// TIA Portal V15.1 export
// export: Created 2024-06-21T08:41:02.0781303Z, ExportSetting WithDefaults, DisplayName Totally Integrated Automation Portal, DisplayVersion V15.1 Update 5, DisplayName TIA Portal Openness, DisplayVersion V15.1 Update 5, DisplayName SINAMICS Startdrive Advanced, DisplayVersion V15.1, DisplayName G130, G150, S120, S150, SINAMICS MV, S210, DisplayVersion V15.1, DisplayName G110M, G120, G120C, G120D, G120P, DisplayVersion V15.1, DisplayName STEP 7 Professional, DisplayVersion V15.1 Update 5, DisplayName STEP 7 Safety, DisplayVersion V15.1, DisplayName WinCC Professional, DisplayVersion V15.1 Update 5, DisplayName SIMATIC Visualization Architect, DisplayVersion V15.1
FUNCTION_BLOCK "LMovFnc3Pos2S"   // FB2192, FBD
TITLE = LMovFnc3Pos2S
{ S7_Optimized_Access := 'TRUE' }
VERSION : 0.1
// =============================================================================
// This module will be used for the steering of a three Position movement wit 2 speed
// It will get the commands from different Modes, evaluate the status of the 
// Interlock and give the command to the Actuator or direct to simple outputs.
// =============================================================================
// stored: AutoNumber false, IsIECCheckEnabled false, IsRetainMemResEnabled false, MemoryReserve 100, SetENOAutomatically False, UDAEnableTagReadback false
   VAR_INPUT
      I_Pos1 { ExternalAccessible := 'False'; ExternalVisible := 'False'; ExternalWritable := 'False'} : Bool;   // Position 1 Detection or Summary
      I_Pos2 { ExternalAccessible := 'False'; ExternalVisible := 'False'; ExternalWritable := 'False'} : Bool;   // Position 2 Detection or Summary
      I_Pos3 { ExternalAccessible := 'False'; ExternalVisible := 'False'; ExternalWritable := 'False'} : Bool;   // Position 3 Detection or Summary
      I_SlowPos1 { ExternalAccessible := 'False'; ExternalVisible := 'False'; ExternalWritable := 'False'} : Bool;   // Slow Position 1 Detection
      I_SlowPos2 { ExternalAccessible := 'False'; ExternalVisible := 'False'; ExternalWritable := 'False'} : Bool;   // Slow Position 2 Detection
      I_SlowPos3 { ExternalAccessible := 'False'; ExternalVisible := 'False'; ExternalWritable := 'False'} : Bool;   // Slow Position 3 Detection
      I_PBSet { ExternalAccessible := 'False'; ExternalVisible := 'False'; ExternalWritable := 'False'} : Bool;   // Push button for Set direction (used in manual with button OP panels )
      I_PBReset { ExternalAccessible := 'False'; ExternalVisible := 'False'; ExternalWritable := 'False'} : Bool;   // Push button for Reset direction (used in manual with Pushbutton OP panels)
      I_Pos1Begin { ExternalAccessible := 'False'; ExternalVisible := 'False'; ExternalWritable := 'False'} : Bool;   // Request Pos 1 Function Begin
      I_Pos2Begin { ExternalAccessible := 'False'; ExternalVisible := 'False'; ExternalWritable := 'False'} : Bool;   // Request Pos 2 Function Begin
      I_Pos3Begin { ExternalAccessible := 'False'; ExternalVisible := 'False'; ExternalWritable := 'False'} : Bool;   // Request Pos 3 Function Begin
      I_SetIntlkOK { ExternalAccessible := 'False'; ExternalVisible := 'False'; ExternalWritable := 'False'} : Bool;   // Interlock Set Ok
      I_ResIntlkOK { ExternalAccessible := 'False'; ExternalVisible := 'False'; ExternalWritable := 'False'} : Bool;   // Interlock Reset Ok
      I_SafetyOk { ExternalAccessible := 'False'; ExternalVisible := 'False'; ExternalWritable := 'False'} : Bool;   // Safety ok
      I_HardwareOk { ExternalAccessible := 'False'; ExternalVisible := 'False'; ExternalWritable := 'False'} : Bool;   // Safety Ok / Hardware Ok
   END_VAR
   VAR_OUTPUT
      O_CmdSetHighSpeed { ExternalAccessible := 'False'; ExternalVisible := 'False'; ExternalWritable := 'False'} : Bool;   // Command to Activate Set movement
      O_CmdResHighSpeed { ExternalAccessible := 'False'; ExternalVisible := 'False'; ExternalWritable := 'False'} : Bool;   // Command to Activate Reset movement
      O_CmdSetLowSpeed { ExternalAccessible := 'False'; ExternalVisible := 'False'; ExternalWritable := 'False'} : Bool;   // Command to Activate Slow Set movement
      O_CmdResLowSpeed { ExternalAccessible := 'False'; ExternalVisible := 'False'; ExternalWritable := 'False'} : Bool;   // Command to Activate Slow Reset movement
      O_CmdPos1 { ExternalAccessible := 'False'; ExternalVisible := 'False'; ExternalWritable := 'False'} : Bool;   // Command to activate Set movement / Command to Activate Pos1 movement
      O_CmdPos2 { ExternalAccessible := 'False'; ExternalVisible := 'False'; ExternalWritable := 'False'} : Bool;   // Command to activate Set movement / Command to Activate Pos2 movement
      O_CmdPos3 { ExternalAccessible := 'False'; ExternalVisible := 'False'; ExternalWritable := 'False'} : Bool;   // Command to activate Reset movement / Command to Activate Pos3 movement
      O_FuncRunning { ExternalAccessible := 'False'; ExternalVisible := 'False'; ExternalWritable := 'False'} : Bool;   // Signal that the function is running
      O_FuncBusyTM { ExternalAccessible := 'False'; ExternalVisible := 'False'; ExternalWritable := 'False'} : Bool;   // Memory Signal that the function is busy
      O_Pos1Finished { ExternalAccessible := 'False'; ExternalVisible := 'False'; ExternalWritable := 'False'} : Bool;   // Position1 Finished
      O_Pos2Finished { ExternalAccessible := 'False'; ExternalVisible := 'False'; ExternalWritable := 'False'} : Bool;   // Position2 Finished
      O_Pos3Finished { ExternalAccessible := 'False'; ExternalVisible := 'False'; ExternalWritable := 'False'} : Bool;   // Position3 Finished
      O_IntlkSetAlm { ExternalAccessible := 'False'; ExternalVisible := 'False'; ExternalWritable := 'False'} : Bool;   // Alarm Interlock Set
      O_IntlkResAlm { ExternalAccessible := 'False'; ExternalVisible := 'False'; ExternalWritable := 'False'} : Bool;   // Alarm Interlock Reset
      O_FuncIsSelInMan { ExternalAccessible := 'False'; ExternalVisible := 'False'; ExternalWritable := 'False'} : Bool;   // The function is Selected in manual Mode
      O_LED { ExternalAccessible := 'False'; ExternalVisible := 'False'; ExternalWritable := 'False'} : Bool;   // LED - Indication
      O_AlarmABCondition { ExternalAccessible := 'False'; ExternalVisible := 'False'; ExternalWritable := 'False'} : Bool;   // Alarms AB condition
   END_VAR
   VAR_IN_OUT
      IO_Modes : "Modes";   // Modes
      H_HMI : "H_HMI";   // Animation
      H_MovFnc3Pos2S : "H_MovFnc3Pos";   // Animation
      H_FncSelInHMI { ExternalAccessible := 'False'; ExternalVisible := 'False'; ExternalWritable := 'False'} : Bool;   // This function is Selected to run from HMI
      C_AlarmResetUsed { ExternalAccessible := 'False'; ExternalVisible := 'False'; ExternalWritable := 'False'} : Bool;   // If true, the alrms will be stored untill Reseted
      C_EnableMemBegin { ExternalAccessible := 'False'; ExternalVisible := 'False'; ExternalWritable := 'False'} : Bool;   // Enable memory Begin (Command request is memorised until pos reached)
      C_EnIntlkAlm { ExternalAccessible := 'False'; ExternalVisible := 'False'; ExternalWritable := 'False'} : Bool := TRUE;   // Enable Interlock Alarm
      C_ForceManual { ExternalAccessible := 'False'; ExternalVisible := 'False'; ExternalWritable := 'False'} : Bool := FALSE;   // Force Manual
   END_VAR
   VAR
      ResetAlarm { ExternalAccessible := 'False'; ExternalVisible := 'False'; ExternalWritable := 'False'} : Bool;   // Reset Alarm Memory
      BeginPos1Req { ExternalAccessible := 'False'; ExternalVisible := 'False'; ExternalWritable := 'False'} : Bool;   // Request Pos 1 Function Begin
      BeginPos2Req { ExternalAccessible := 'False'; ExternalVisible := 'False'; ExternalWritable := 'False'} : Bool;   // Request Pos 2 Function Begin
      BeginPos3Req { ExternalAccessible := 'False'; ExternalVisible := 'False'; ExternalWritable := 'False'} : Bool;   // Request Pos 3 Function Begin
      CmdSet { ExternalAccessible := 'False'; ExternalVisible := 'False'; ExternalWritable := 'False'} : Bool;   // Command set
      CmdSetSl { ExternalAccessible := 'False'; ExternalVisible := 'False'; ExternalWritable := 'False'} : Bool;   // Command to Activate Slow Set movement
      CmdSetRequest { ExternalAccessible := 'False'; ExternalVisible := 'False'; ExternalWritable := 'False'} : Bool;   // Set Command request to Activate the Interlock
      CmdRes { ExternalAccessible := 'False'; ExternalVisible := 'False'; ExternalWritable := 'False'} : Bool;   // Command Reset
      CmdResSl { ExternalAccessible := 'False'; ExternalVisible := 'False'; ExternalWritable := 'False'} : Bool;   // Command to Activate Slow Reset movement
      CmdResRequest { ExternalAccessible := 'False'; ExternalVisible := 'False'; ExternalWritable := 'False'} : Bool;   // Reset Command request to Activate the Interlock
   END_VAR
   VAR RETAIN
      BetweenPos1Pos2 { ExternalAccessible := 'False'; ExternalVisible := 'False'; ExternalWritable := 'False'} : Bool;   // Table Between Pos 1 And 2
      BetweenPos1Pos2Set { ExternalAccessible := 'False'; ExternalVisible := 'False'; ExternalWritable := 'False'} : Bool;   // Table Between Pos 1 And 2 Set
      BetweenPos1Pos2Res { ExternalAccessible := 'False'; ExternalVisible := 'False'; ExternalWritable := 'False'} : Bool;   // Table Between Pos 1 And 2 Reset
      BetweenPos2Pos3 { ExternalAccessible := 'False'; ExternalVisible := 'False'; ExternalWritable := 'False'} : Bool;   // Table Between Pos 2 And 3
      BetweenPos2Pos3Set { ExternalAccessible := 'False'; ExternalVisible := 'False'; ExternalWritable := 'False'} : Bool;   // Table Between Pos 2 And 3 Set
      BetweenPos2Pos3Res { ExternalAccessible := 'False'; ExternalVisible := 'False'; ExternalWritable := 'False'} : Bool;   // Table Between Pos 2 And 3 Reset
   END_VAR
   VAR
      Pos2SetReached { ExternalAccessible := 'False'; ExternalVisible := 'False'; ExternalWritable := 'False'} : Bool;   // Position 2 Set Reached
      P_CmdSetRequest { ExternalAccessible := 'False'; ExternalVisible := 'False'; ExternalWritable := 'False'} : Bool;   // Cmd Request Set Pos Trig
      Pos2ResReached { ExternalAccessible := 'False'; ExternalVisible := 'False'; ExternalWritable := 'False'} : Bool;   // Position 2 Reset Reached
      P_CmdResRequest { ExternalAccessible := 'False'; ExternalVisible := 'False'; ExternalWritable := 'False'} : Bool;   // Cmd Request Res Pos Trig
      CmdPos1 { ExternalAccessible := 'False'; ExternalVisible := 'False'; ExternalWritable := 'False'} : Bool;   // Command to activate Set movement / Command to Activate Pos1 movement
      CmdPos2 { ExternalAccessible := 'False'; ExternalVisible := 'False'; ExternalWritable := 'False'} : Bool;   // Command to activate Set movement / Command to Activate Pos2 movement
      CmdPos3 { ExternalAccessible := 'False'; ExternalVisible := 'False'; ExternalWritable := 'False'} : Bool;   // Command to activate Reset movement / Command to Activate Pos3 movement
      IntlkSetAlm { ExternalAccessible := 'False'; ExternalVisible := 'False'; ExternalWritable := 'False'} : Bool;   // Alarm Interlock Set
      IntlkResAlm { ExternalAccessible := 'False'; ExternalVisible := 'False'; ExternalWritable := 'False'} : Bool;   // Alarm Interlock Reset
      IntlkSetAlmCond { ExternalAccessible := 'False'; ExternalVisible := 'False'; ExternalWritable := 'False'} : Bool;   // Alarm Interlock Set condition
      IntlkResAlmCond { ExternalAccessible := 'False'; ExternalVisible := 'False'; ExternalWritable := 'False'} : Bool;   // Alarm Interlock Reset condition
      FuncRunning { ExternalAccessible := 'False'; ExternalVisible := 'False'; ExternalWritable := 'False'} : Bool;   // Function is running
      FuncBusyTM { ExternalAccessible := 'False'; ExternalVisible := 'False'; ExternalWritable := 'False'} : Bool;   // Memory Signal that the function is busy
      Edge { ExternalAccessible := 'False'; ExternalVisible := 'False'; ExternalWritable := 'False'} : Array[1..5] of Bool;   // Edge
      AlarmTimer { ExternalAccessible := 'False'; ExternalVisible := 'False'; ExternalWritable := 'False'} : "LTimer";
      AlmFilterResult { ExternalAccessible := 'False'; ExternalVisible := 'False'; ExternalWritable := 'False'} : Bool;
   END_VAR
   VAR_TEMP   // added for the SCL form of the ladder/FBD networks
      _w1 : Bool;
      _w2 : Bool;
      _w3 : Bool;
      _w4 : Bool;
   END_VAR
BEGIN

REGION Network 1: **** 2.2 - Alarms - Alarm Generation **** Alarm Filter
   // Alarm Filter
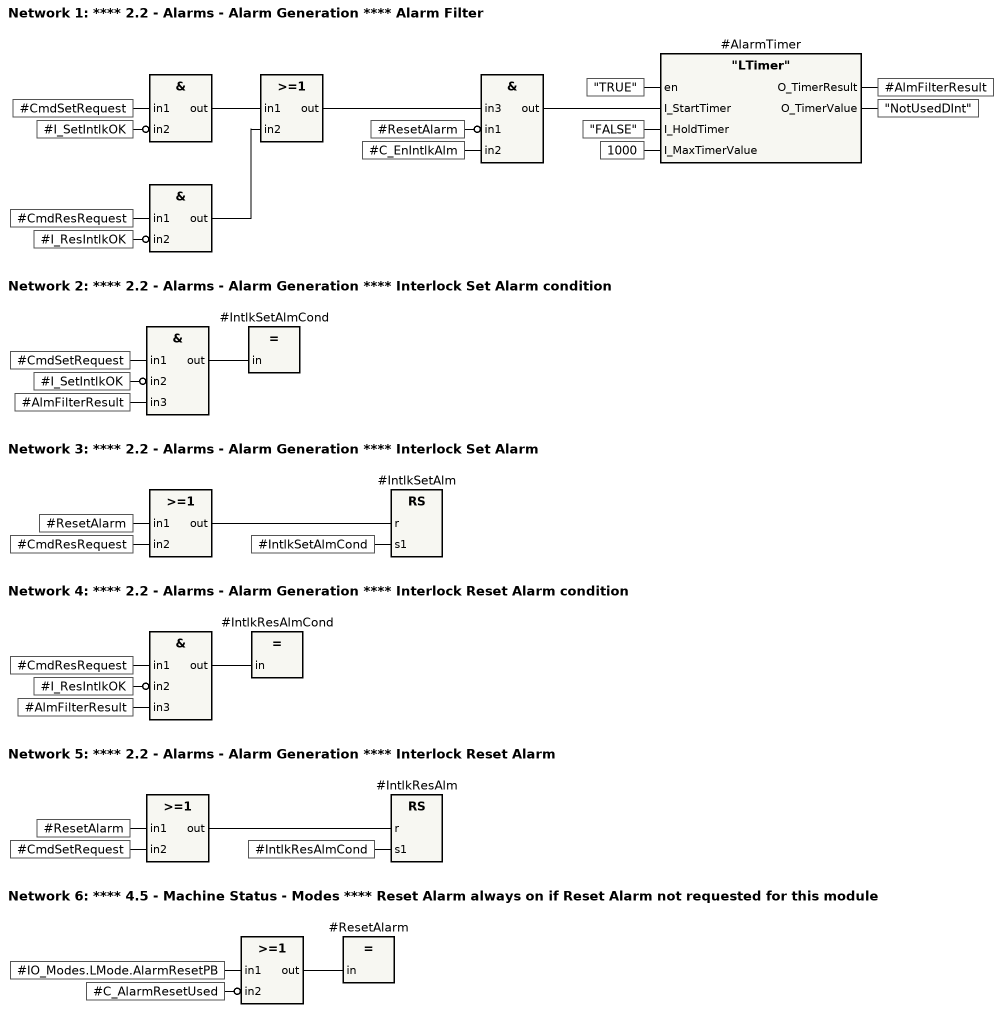
   IF "TRUE" THEN
       #AlarmTimer(I_StartTimer := ((#CmdSetRequest AND NOT #I_SetIntlkOK) OR (#CmdResRequest AND NOT #I_ResIntlkOK)) AND NOT #ResetAlarm AND #C_EnIntlkAlm,   // "LTimer"
                   I_HoldTimer := "FALSE",
                   I_MaxTimerValue := 1000,
                   O_TimerResult => #AlmFilterResult,
                   O_TimerValue => "NotUsedDInt");
   END_IF;
END_REGION

REGION Network 2: **** 2.2 - Alarms - Alarm Generation **** Interlock Set Alarm condition
   // Interlock Set Alarm condition
   #IntlkSetAlmCond := #CmdSetRequest AND NOT #I_SetIntlkOK AND #AlmFilterResult;
END_REGION

REGION Network 3: **** 2.2 - Alarms - Alarm Generation **** Interlock Set Alarm
   // Interlock Set Alarm
   IF #ResetAlarm OR #CmdResRequest THEN
       #IntlkSetAlm := FALSE;   // RS flip-flop
   END_IF;
   IF #IntlkSetAlmCond THEN #IntlkSetAlm := TRUE; END_IF;
END_REGION

REGION Network 4: **** 2.2 - Alarms - Alarm Generation **** Interlock Reset Alarm condition
   // Interlock Reset Alarm condition
   #IntlkResAlmCond := #CmdResRequest AND NOT #I_ResIntlkOK AND #AlmFilterResult;
END_REGION

REGION Network 5: **** 2.2 - Alarms - Alarm Generation **** Interlock Reset Alarm
   // Interlock Reset Alarm
   IF #ResetAlarm OR #CmdSetRequest THEN
       #IntlkResAlm := FALSE;   // RS flip-flop
   END_IF;
   IF #IntlkResAlmCond THEN #IntlkResAlm := TRUE; END_IF;
END_REGION

REGION Network 6: **** 4.5 - Machine Status - Modes **** Reset Alarm always on if Reset Alarm not requested for this module
   // Reset Alarm always on if Reset Alarm not requested for this module
   #ResetAlarm := #IO_Modes.LMode.AlarmResetPB OR NOT #C_AlarmResetUsed;
END_REGION

REGION Network 7: **** 4.6 - Machine Status - Indication **** Icon Animation
   // Icon Animation
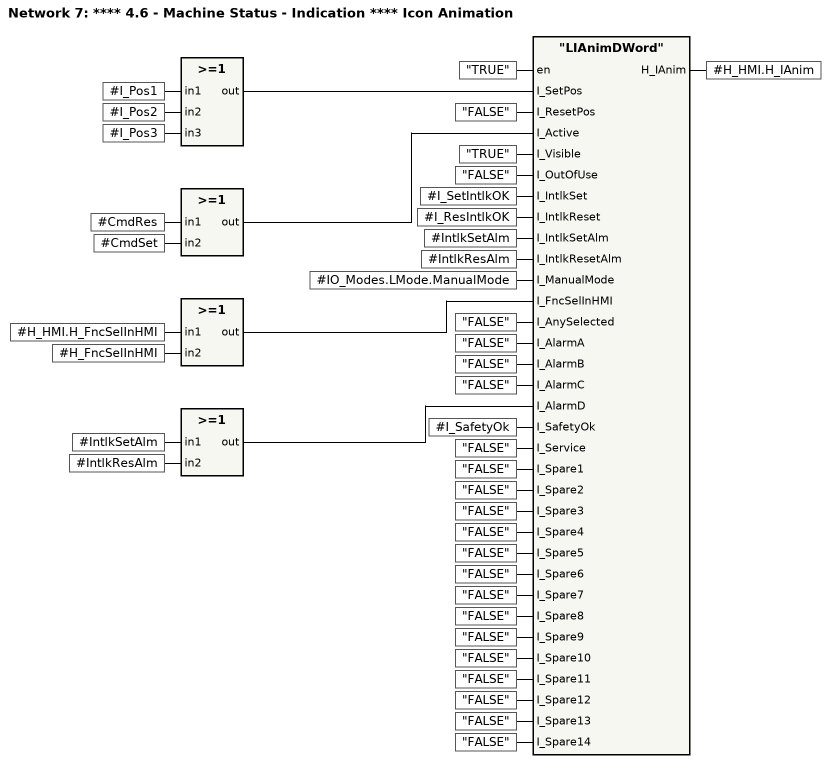
   IF "TRUE" THEN
       "LIAnimDWord"(I_SetPos := #I_Pos1 OR #I_Pos2 OR #I_Pos3,
                     I_ResetPos := "FALSE",
                     I_Active := #CmdRes OR #CmdSet,
                     I_Visible := "TRUE",
                     I_OutOfUse := "FALSE",
                     I_IntlkSet := #I_SetIntlkOK,
                     I_IntlkReset := #I_ResIntlkOK,
                     I_IntlkSetAlm := #IntlkSetAlm,
                     I_IntlkResetAlm := #IntlkResAlm,
                     I_ManualMode := #IO_Modes.LMode.ManualMode,
                     I_FncSelInHMI := #H_HMI.H_FncSelInHMI OR #H_FncSelInHMI,
                     I_AnySelected := "FALSE",
                     I_AlarmA := "FALSE",
                     I_AlarmB := "FALSE",
                     I_AlarmC := "FALSE",
                     I_AlarmD := #IntlkSetAlm OR #IntlkResAlm,
                     I_SafetyOk := #I_SafetyOk,
                     I_Service := "FALSE",
                     I_Spare1 := "FALSE",
                     I_Spare2 := "FALSE",
                     I_Spare3 := "FALSE",
                     I_Spare4 := "FALSE",
                     I_Spare5 := "FALSE",
                     I_Spare6 := "FALSE",
                     I_Spare7 := "FALSE",
                     I_Spare8 := "FALSE",
                     I_Spare9 := "FALSE",
                     I_Spare10 := "FALSE",
                     I_Spare11 := "FALSE",
                     I_Spare12 := "FALSE",
                     I_Spare13 := "FALSE",
                     I_Spare14 := "FALSE",
                     H_IAnim => #H_HMI.H_IAnim);
   END_IF;
END_REGION

REGION Network 8: **** 4.6 - Machine Status - Indication **** Animation
   // Animation
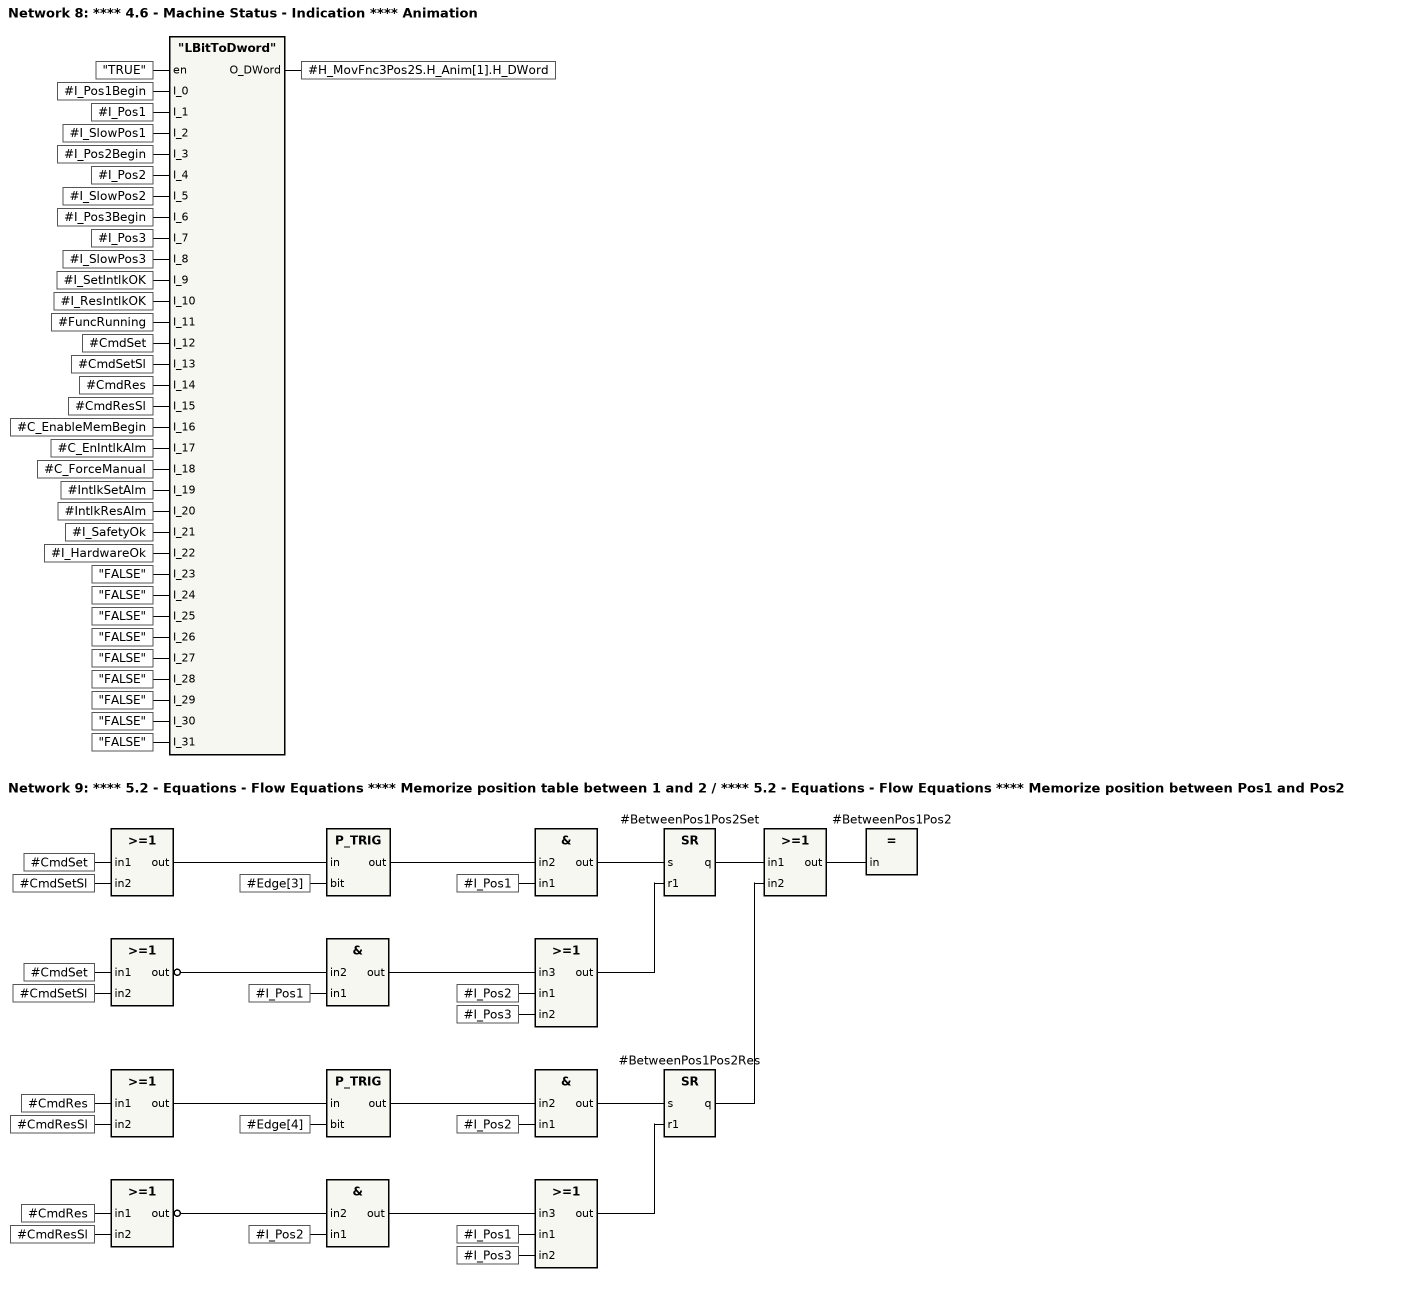
   IF "TRUE" THEN
       "LBitToDword"(I_0 := #I_Pos1Begin,
                     I_1 := #I_Pos1,
                     I_2 := #I_SlowPos1,
                     I_3 := #I_Pos2Begin,
                     I_4 := #I_Pos2,
                     I_5 := #I_SlowPos2,
                     I_6 := #I_Pos3Begin,
                     I_7 := #I_Pos3,
                     I_8 := #I_SlowPos3,
                     I_9 := #I_SetIntlkOK,
                     I_10 := #I_ResIntlkOK,
                     I_11 := #FuncRunning,
                     I_12 := #CmdSet,
                     I_13 := #CmdSetSl,
                     I_14 := #CmdRes,
                     I_15 := #CmdResSl,
                     I_16 := #C_EnableMemBegin,
                     I_17 := #C_EnIntlkAlm,
                     I_18 := #C_ForceManual,
                     I_19 := #IntlkSetAlm,
                     I_20 := #IntlkResAlm,
                     I_21 := #I_SafetyOk,
                     I_22 := #I_HardwareOk,
                     I_23 := "FALSE",
                     I_24 := "FALSE",
                     I_25 := "FALSE",
                     I_26 := "FALSE",
                     I_27 := "FALSE",
                     I_28 := "FALSE",
                     I_29 := "FALSE",
                     I_30 := "FALSE",
                     I_31 := "FALSE",
                     O_DWord => #H_MovFnc3Pos2S.H_Anim[1].H_DWord);
   END_IF;
END_REGION

REGION Network 9: **** 5.2 - Equations - Flow Equations **** Memorize position table between 1 and 2 / **** 5.2 - Equations - Flow Equations **** Memorize position between Pos1 and Pos2
   // Memorize Position table between 1 and 2
   #_w1 := #CmdSet OR #CmdSetSl;
   #_w2 := #_w1 AND NOT #Edge[3];   // rising edge
   #Edge[3] := #_w1;
   IF #_w2 AND #I_Pos1 THEN
       #BetweenPos1Pos2Set := TRUE;   // SR flip-flop
   END_IF;
   IF (NOT (#CmdSet OR #CmdSetSl) AND #I_Pos1) OR #I_Pos2 OR #I_Pos3 THEN
       #BetweenPos1Pos2Set := FALSE;
   END_IF;
   #_w3 := #CmdRes OR #CmdResSl;
   #_w4 := #_w3 AND NOT #Edge[4];   // rising edge
   #Edge[4] := #_w3;
   IF #_w4 AND #I_Pos2 THEN
       #BetweenPos1Pos2Res := TRUE;   // SR flip-flop
   END_IF;
   IF (NOT (#CmdRes OR #CmdResSl) AND #I_Pos2) OR #I_Pos1 OR #I_Pos3 THEN
       #BetweenPos1Pos2Res := FALSE;
   END_IF;
   #BetweenPos1Pos2 := #BetweenPos1Pos2Set OR #BetweenPos1Pos2Res;
END_REGION

REGION Network 10: **** 5.2 - Equations - Flow Equations **** Memorize position between 2 and 3 / **** 5.2 - Equations - Flow Equations **** Memorize position between Pos2 and Pos3
   // Memorize Position table  2 and 3
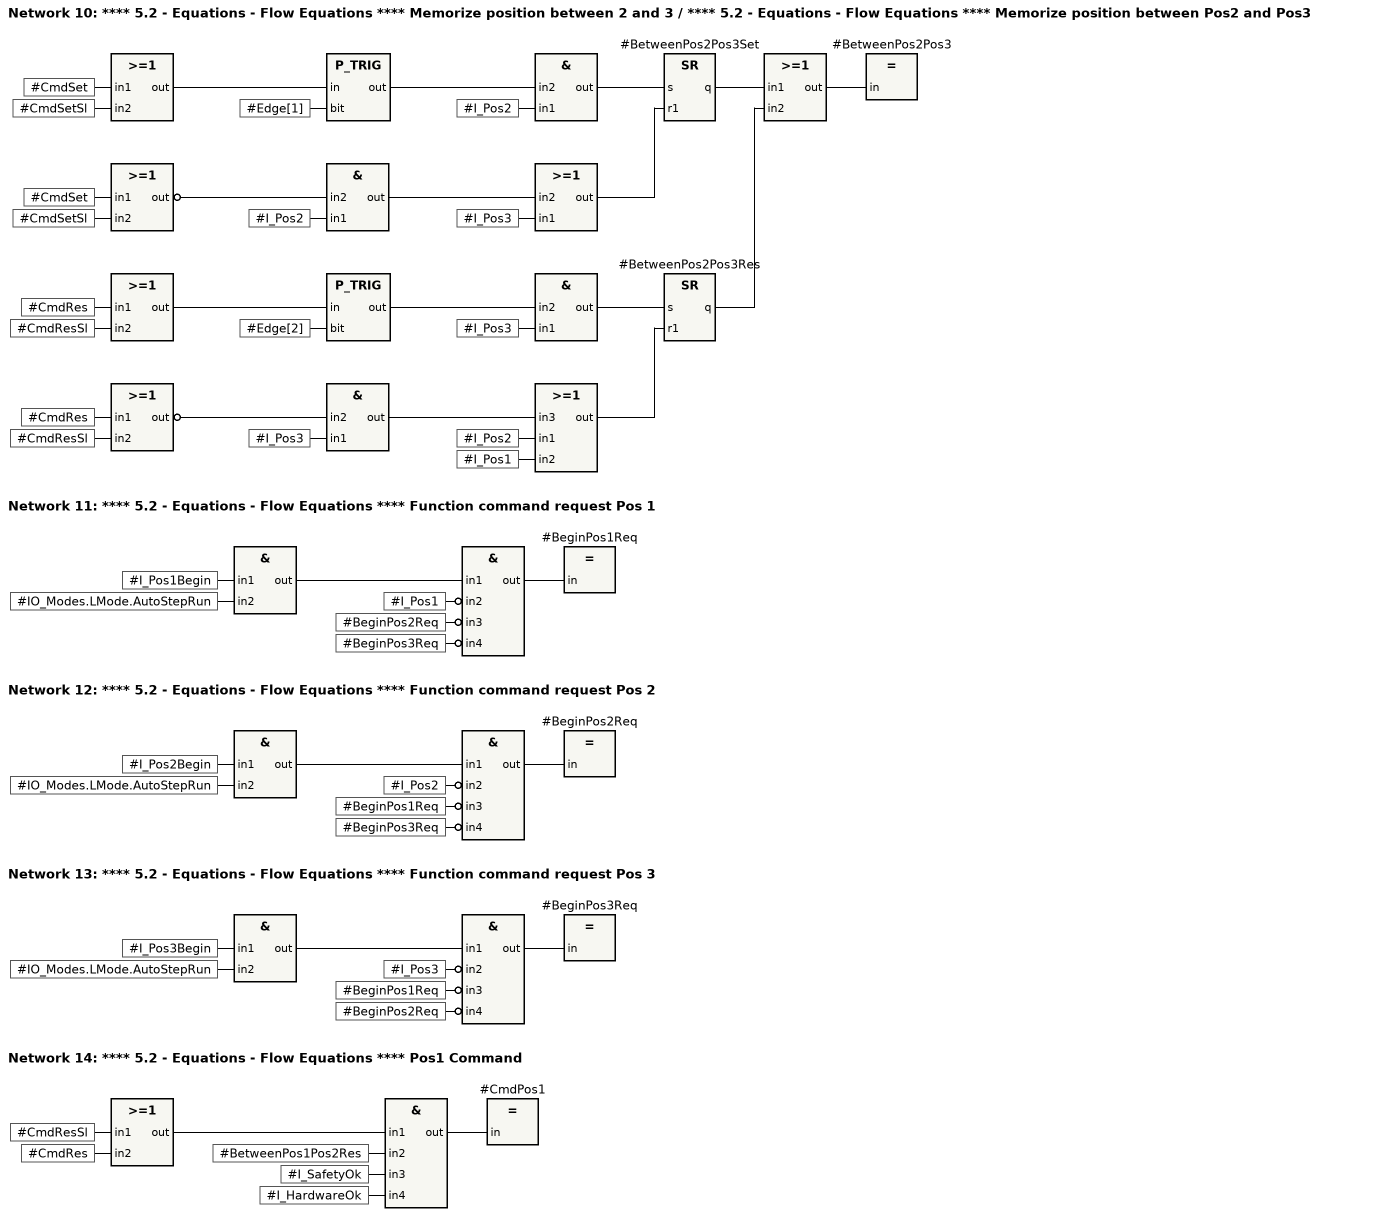
   #_w1 := #CmdSet OR #CmdSetSl;
   #_w2 := #_w1 AND NOT #Edge[1];   // rising edge
   #Edge[1] := #_w1;
   IF #_w2 AND #I_Pos2 THEN
       #BetweenPos2Pos3Set := TRUE;   // SR flip-flop
   END_IF;
   IF (NOT (#CmdSet OR #CmdSetSl) AND #I_Pos2) OR #I_Pos3 THEN #BetweenPos2Pos3Set := FALSE; END_IF;
   #_w3 := #CmdRes OR #CmdResSl;
   #_w4 := #_w3 AND NOT #Edge[2];   // rising edge
   #Edge[2] := #_w3;
   IF #_w4 AND #I_Pos3 THEN
       #BetweenPos2Pos3Res := TRUE;   // SR flip-flop
   END_IF;
   IF (NOT (#CmdRes OR #CmdResSl) AND #I_Pos3) OR #I_Pos2 OR #I_Pos1 THEN
       #BetweenPos2Pos3Res := FALSE;
   END_IF;
   #BetweenPos2Pos3 := #BetweenPos2Pos3Set OR #BetweenPos2Pos3Res;
END_REGION

REGION Network 11: **** 5.2 - Equations - Flow Equations **** Function command request Pos 1
   // Function command request Pos 1
   #BeginPos1Req := #I_Pos1Begin AND #IO_Modes.LMode.AutoStepRun AND NOT #I_Pos1 AND NOT #BeginPos2Req AND NOT #BeginPos3Req;
END_REGION

REGION Network 12: **** 5.2 - Equations - Flow Equations **** Function command request Pos 2
   // Function command request Pos 2
   #BeginPos2Req := #I_Pos2Begin AND #IO_Modes.LMode.AutoStepRun AND NOT #I_Pos2 AND NOT #BeginPos1Req AND NOT #BeginPos3Req;
END_REGION

REGION Network 13: **** 5.2 - Equations - Flow Equations **** Function command request Pos 3
   // Function command request Pos 3
   #BeginPos3Req := #I_Pos3Begin AND #IO_Modes.LMode.AutoStepRun AND NOT #I_Pos3 AND NOT #BeginPos1Req AND NOT #BeginPos2Req;
END_REGION

REGION Network 14: **** 5.2 - Equations - Flow Equations **** Pos1 Command
   // Pos1 Command
   #CmdPos1 := (#CmdResSl OR #CmdRes) AND #BetweenPos1Pos2Res AND #I_SafetyOk AND #I_HardwareOk;
END_REGION

REGION Network 15: **** 5.2 - Equations - Flow Equations **** Pos2 Command
   // Pos2 Command
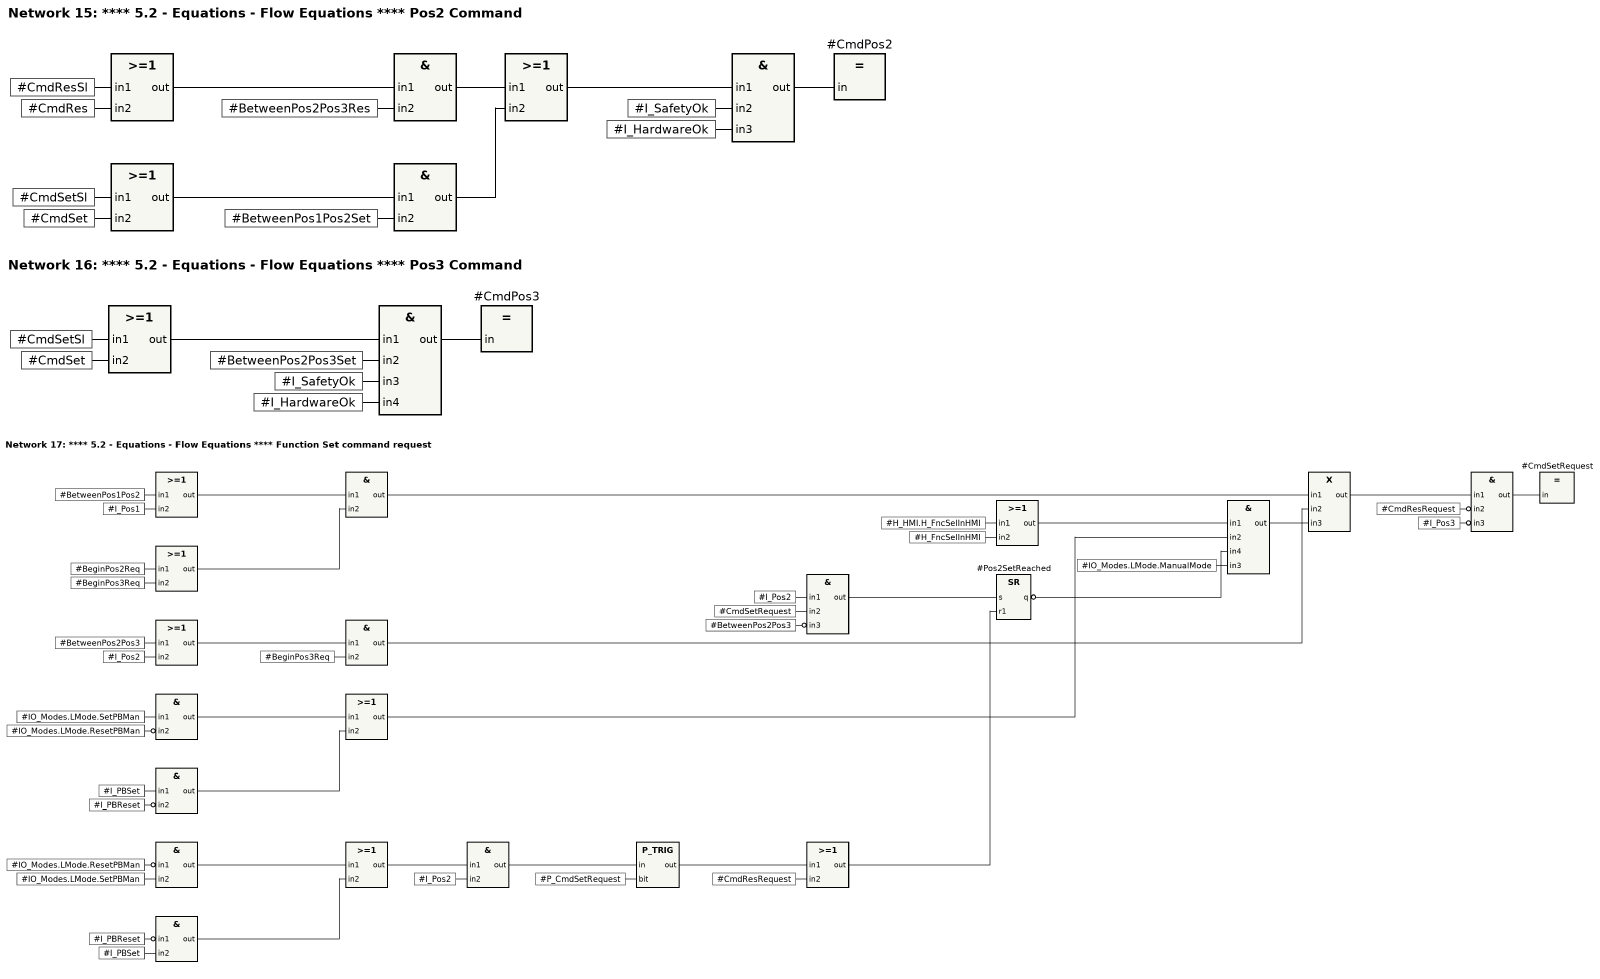
   #CmdPos2 := (((#CmdResSl OR #CmdRes) AND #BetweenPos2Pos3Res) OR ((#CmdSetSl OR #CmdSet) AND #BetweenPos1Pos2Set)) AND #I_SafetyOk AND #I_HardwareOk;
END_REGION

REGION Network 16: **** 5.2 - Equations - Flow Equations **** Pos3 Command
   // Pos3 Command
   #CmdPos3 := (#CmdSetSl OR #CmdSet) AND #BetweenPos2Pos3Set AND #I_SafetyOk AND #I_HardwareOk;
END_REGION

REGION Network 17: **** 5.2 - Equations - Flow Equations **** Function Set command request
   // Function Set command request
   #_w1 := ((NOT #IO_Modes.LMode.ResetPBMan AND #IO_Modes.LMode.SetPBMan) OR (NOT #I_PBReset AND #I_PBSet)) AND #I_Pos2;
   #_w2 := #_w1 AND NOT #P_CmdSetRequest;   // rising edge
   #P_CmdSetRequest := #_w1;
   IF #I_Pos2 AND #CmdSetRequest AND NOT #BetweenPos2Pos3 THEN
       #Pos2SetReached := TRUE;   // SR flip-flop
   END_IF;
   IF #_w2 OR #CmdResRequest THEN #Pos2SetReached := FALSE; END_IF;
   #CmdSetRequest := (((#BetweenPos1Pos2 OR #I_Pos1) AND (#BeginPos2Req OR #BeginPos3Req)) XOR ((#BetweenPos2Pos3 OR #I_Pos2) AND #BeginPos3Req) XOR ((#H_HMI.H_FncSelInHMI OR #H_FncSelInHMI) AND ((#IO_Modes.LMode.SetPBMan AND NOT #IO_Modes.LMode.ResetPBMan) OR (#I_PBSet AND NOT #I_PBReset)) AND NOT #Pos2SetReached AND #IO_Modes.LMode.ManualMode)) AND NOT #CmdResRequest AND NOT #I_Pos3;
END_REGION

REGION Network 18: **** 5.2 - Equations - Flow Equations **** Function Reset command request
   // Function Reset command request
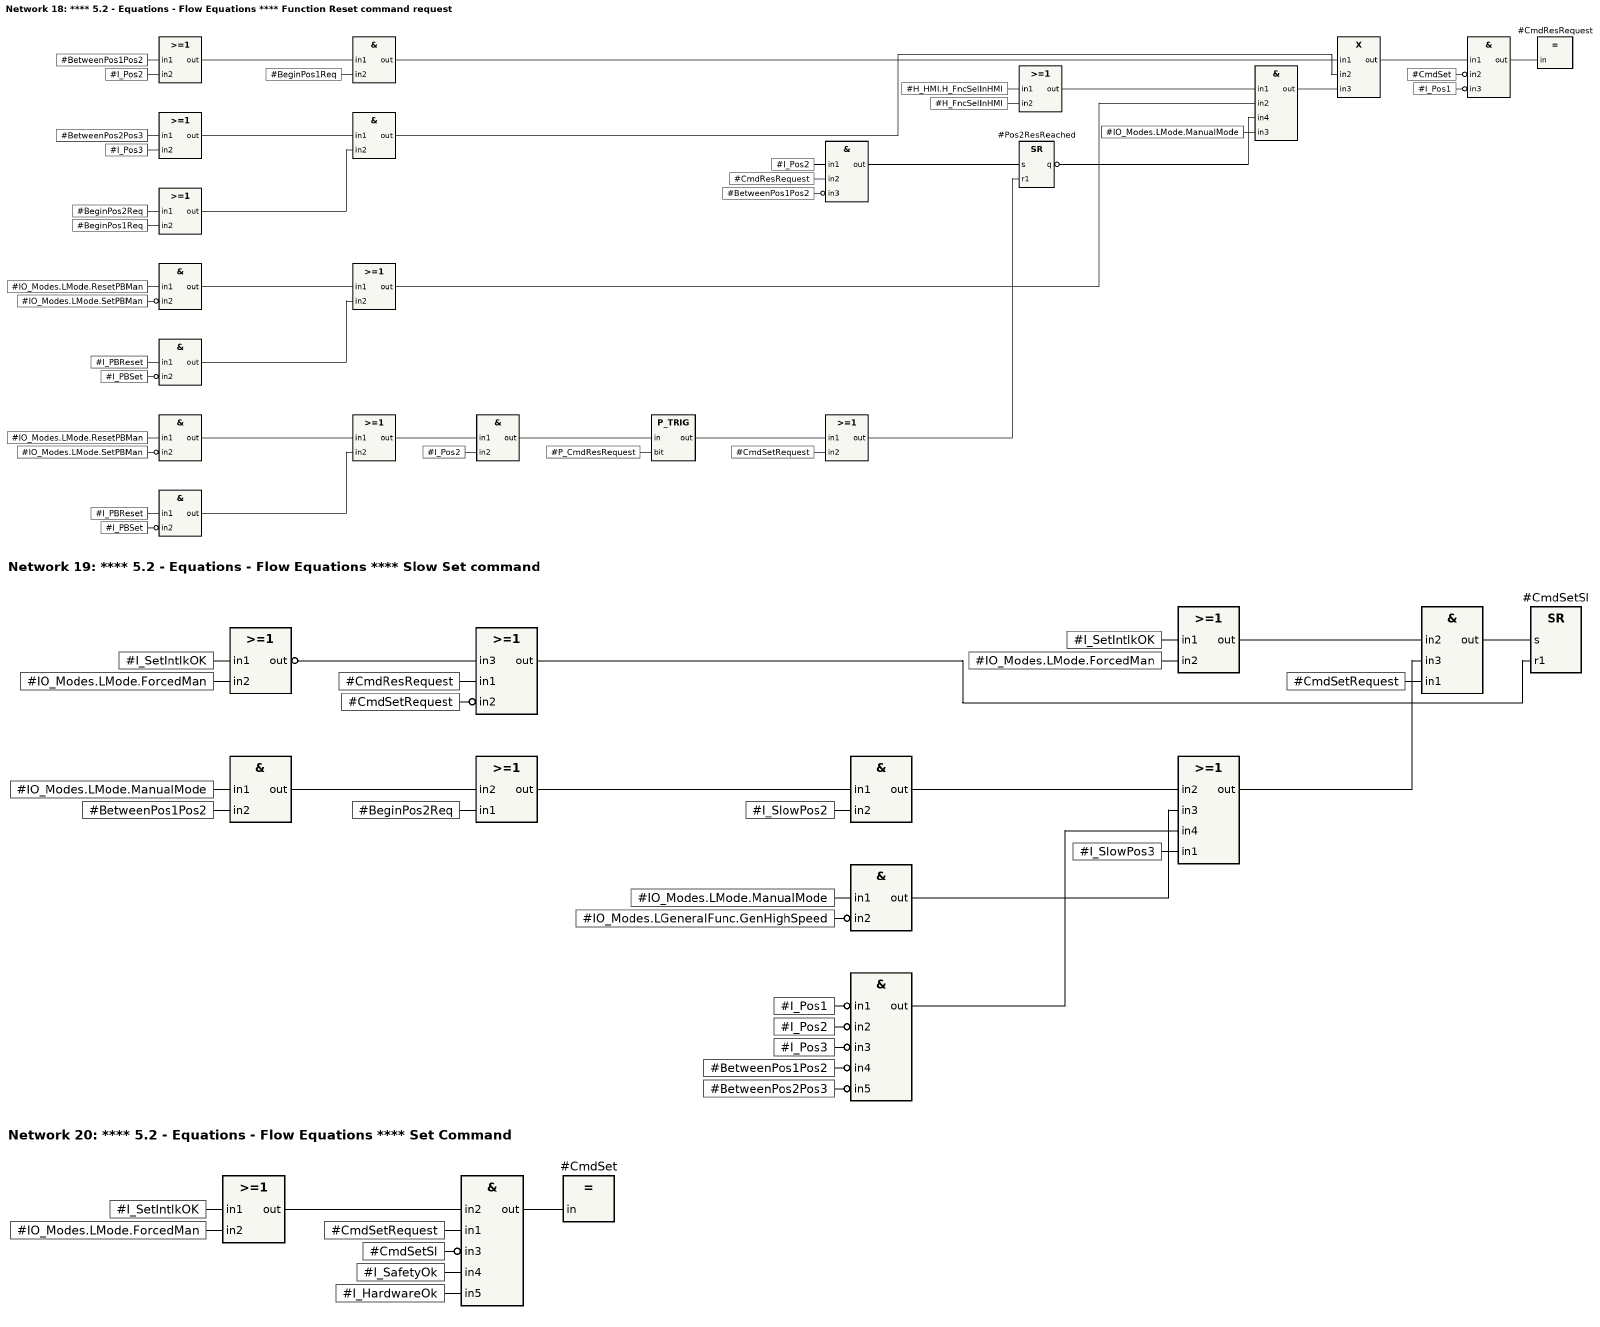
   #_w1 := ((#IO_Modes.LMode.ResetPBMan AND NOT #IO_Modes.LMode.SetPBMan) OR (#I_PBReset AND NOT #I_PBSet)) AND #I_Pos2;
   #_w2 := #_w1 AND NOT #P_CmdResRequest;   // rising edge
   #P_CmdResRequest := #_w1;
   IF #I_Pos2 AND #CmdResRequest AND NOT #BetweenPos1Pos2 THEN
       #Pos2ResReached := TRUE;   // SR flip-flop
   END_IF;
   IF #_w2 OR #CmdSetRequest THEN #Pos2ResReached := FALSE; END_IF;
   #CmdResRequest := (((#BetweenPos1Pos2 OR #I_Pos2) AND #BeginPos1Req) XOR ((#BetweenPos2Pos3 OR #I_Pos3) AND (#BeginPos2Req OR #BeginPos1Req)) XOR ((#H_HMI.H_FncSelInHMI OR #H_FncSelInHMI) AND ((#IO_Modes.LMode.ResetPBMan AND NOT #IO_Modes.LMode.SetPBMan) OR (#I_PBReset AND NOT #I_PBSet)) AND NOT #Pos2ResReached AND #IO_Modes.LMode.ManualMode)) AND NOT #CmdSet AND NOT #I_Pos1;
END_REGION

REGION Network 19: **** 5.2 - Equations - Flow Equations **** Slow Set command
   // Slow Set command
   IF (#I_SetIntlkOK OR #IO_Modes.LMode.ForcedMan) AND ((((#IO_Modes.LMode.ManualMode AND #BetweenPos1Pos2) OR #BeginPos2Req) AND #I_SlowPos2) OR (#IO_Modes.LMode.ManualMode AND NOT #IO_Modes.LGeneralFunc.GenHighSpeed) OR (NOT #I_Pos1 AND NOT #I_Pos2 AND NOT #I_Pos3 AND NOT #BetweenPos1Pos2 AND NOT #BetweenPos2Pos3) OR #I_SlowPos3) AND #CmdSetRequest THEN
       #CmdSetSl := TRUE;   // SR flip-flop
   END_IF;
   IF NOT (#I_SetIntlkOK OR #IO_Modes.LMode.ForcedMan) OR #CmdResRequest OR NOT #CmdSetRequest THEN
       #CmdSetSl := FALSE;
   END_IF;
END_REGION

REGION Network 20: **** 5.2 - Equations - Flow Equations **** Set Command
   // Set Command
   #CmdSet := (#I_SetIntlkOK OR #IO_Modes.LMode.ForcedMan) AND #CmdSetRequest AND NOT #CmdSetSl AND #I_SafetyOk AND #I_HardwareOk;
END_REGION

REGION Network 21: **** 5.2 - Equations - Flow Equations **** Slow Reset command
   // Slow Reset command
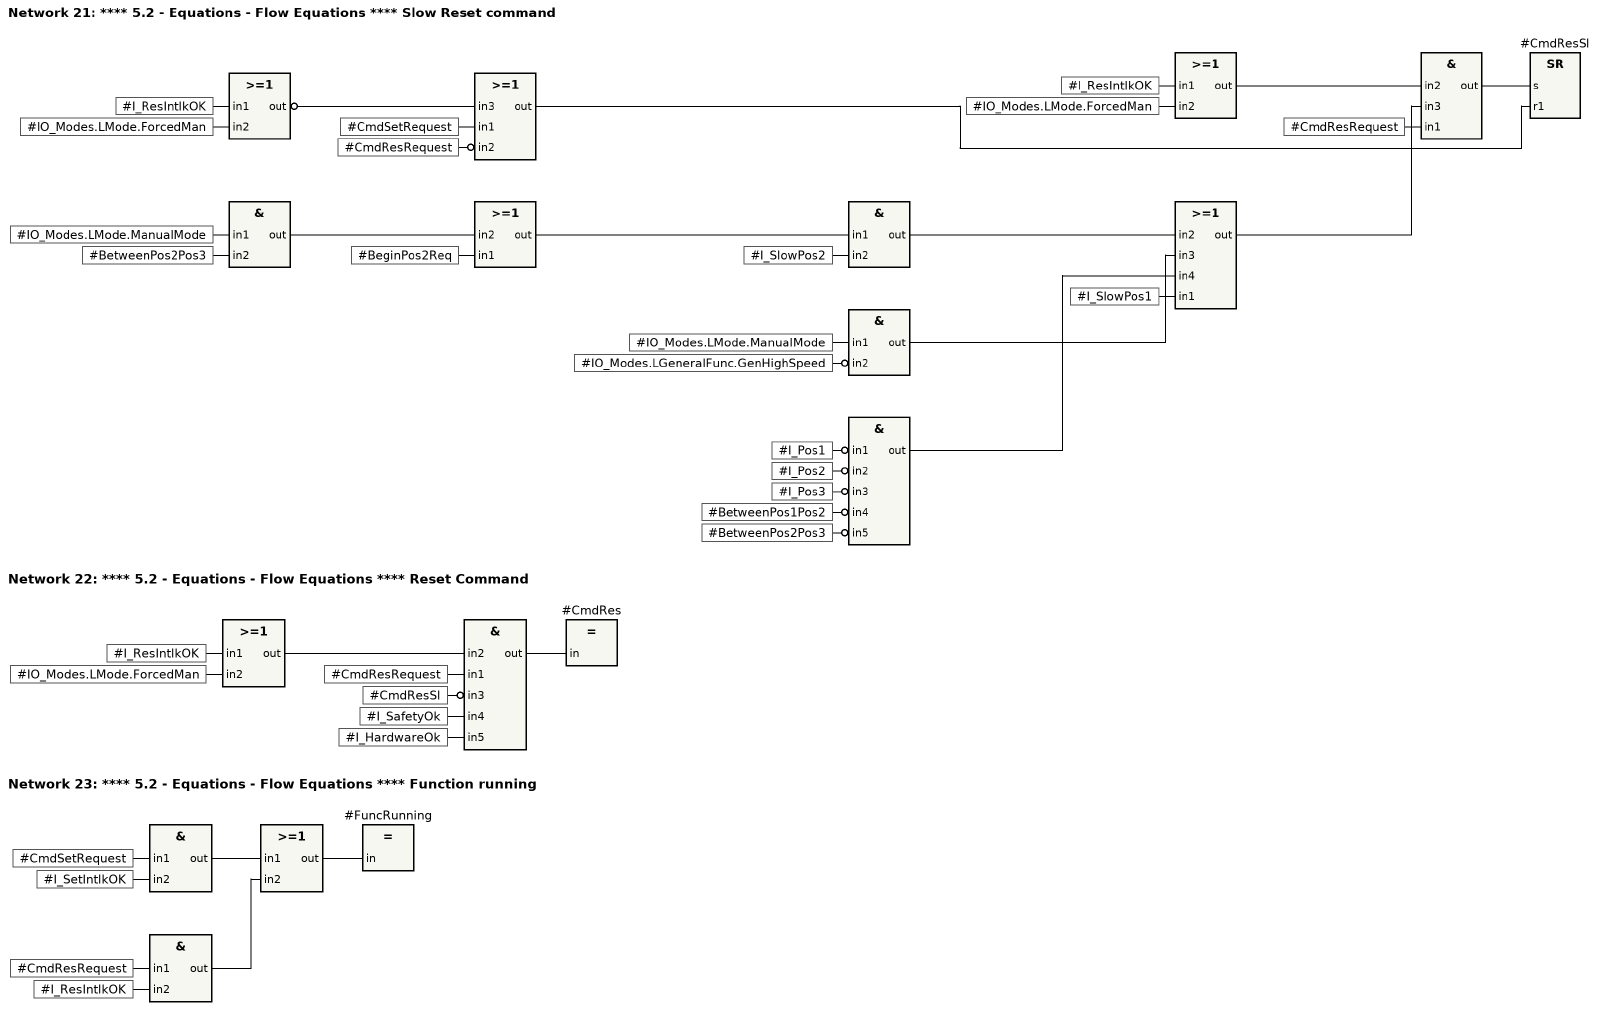
   IF (#I_ResIntlkOK OR #IO_Modes.LMode.ForcedMan) AND ((((#IO_Modes.LMode.ManualMode AND #BetweenPos2Pos3) OR #BeginPos2Req) AND #I_SlowPos2) OR (#IO_Modes.LMode.ManualMode AND NOT #IO_Modes.LGeneralFunc.GenHighSpeed) OR (NOT #I_Pos1 AND NOT #I_Pos2 AND NOT #I_Pos3 AND NOT #BetweenPos1Pos2 AND NOT #BetweenPos2Pos3) OR #I_SlowPos1) AND #CmdResRequest THEN
       #CmdResSl := TRUE;   // SR flip-flop
   END_IF;
   IF NOT (#I_ResIntlkOK OR #IO_Modes.LMode.ForcedMan) OR #CmdSetRequest OR NOT #CmdResRequest THEN
       #CmdResSl := FALSE;
   END_IF;
END_REGION

REGION Network 22: **** 5.2 - Equations - Flow Equations **** Reset Command
   // Reset Command
   #CmdRes := (#I_ResIntlkOK OR #IO_Modes.LMode.ForcedMan) AND #CmdResRequest AND NOT #CmdResSl AND #I_SafetyOk AND #I_HardwareOk;
END_REGION

REGION Network 23: **** 5.2 - Equations - Flow Equations **** Function running
   // Function running
   #FuncRunning := (#CmdSetRequest AND #I_SetIntlkOK) OR (#CmdResRequest AND #I_ResIntlkOK);
END_REGION

REGION Network 24: **** 5.2 - Equations - Flow Equations **** Set Function Running
   // Set Function Running
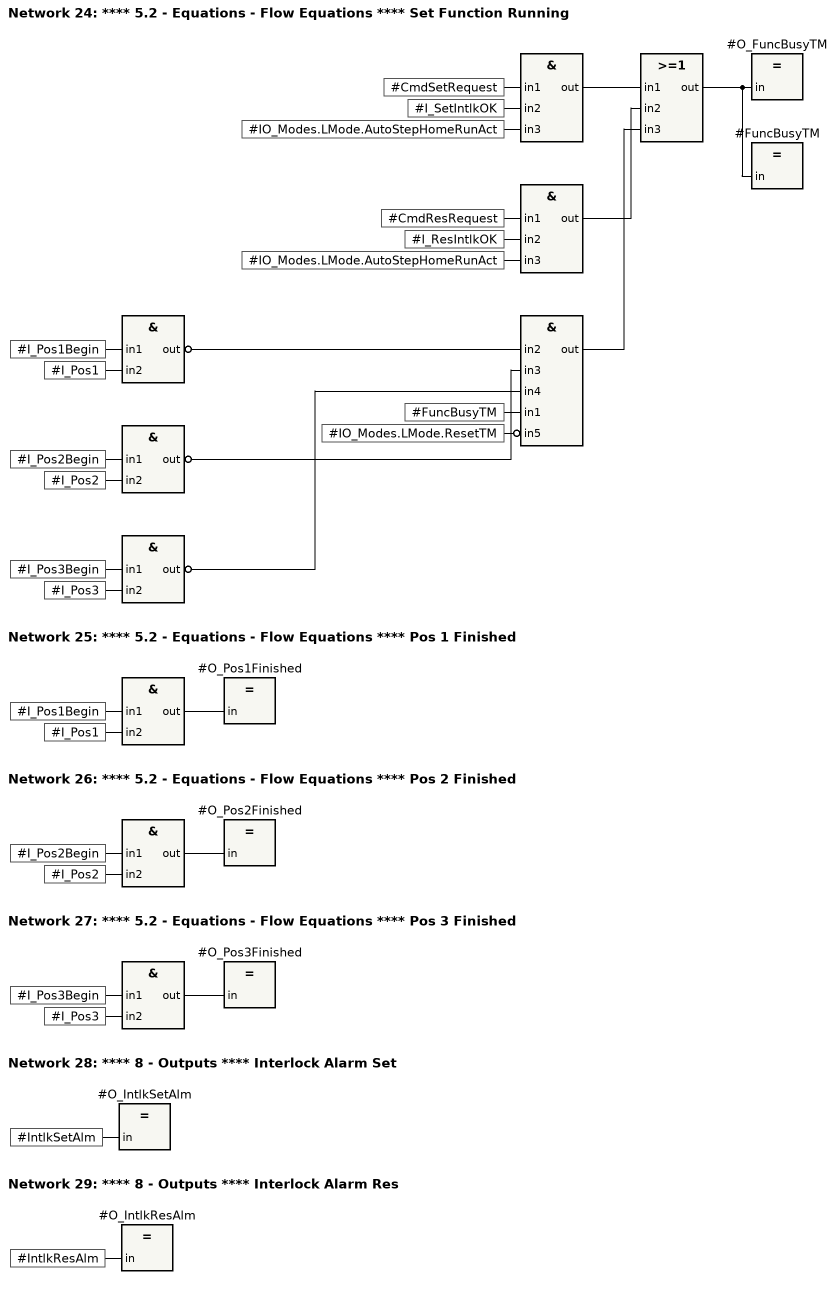
   #O_FuncBusyTM := (#CmdSetRequest AND #I_SetIntlkOK AND #IO_Modes.LMode.AutoStepHomeRunAct) OR (#CmdResRequest AND #I_ResIntlkOK AND #IO_Modes.LMode.AutoStepHomeRunAct) OR (NOT (#I_Pos1Begin AND #I_Pos1) AND NOT (#I_Pos2Begin AND #I_Pos2) AND NOT (#I_Pos3Begin AND #I_Pos3) AND #FuncBusyTM AND NOT #IO_Modes.LMode.ResetTM);
   #FuncBusyTM := #O_FuncBusyTM;
END_REGION

REGION Network 25: **** 5.2 - Equations - Flow Equations **** Pos 1 Finished
   // Pos 1 Finished
   #O_Pos1Finished := #I_Pos1Begin AND #I_Pos1;
END_REGION

REGION Network 26: **** 5.2 - Equations - Flow Equations **** Pos 2 Finished
   // Pos 2 Finished
   #O_Pos2Finished := #I_Pos2Begin AND #I_Pos2;
END_REGION

REGION Network 27: **** 5.2 - Equations - Flow Equations **** Pos 3 Finished
   // Pos 3 Finished
   #O_Pos3Finished := #I_Pos3Begin AND #I_Pos3;
END_REGION

REGION Network 28: **** 8 - Outputs **** Interlock Alarm Set
   // Interlock Alarm Set
   #O_IntlkSetAlm := #IntlkSetAlm;
END_REGION

REGION Network 29: **** 8 - Outputs **** Interlock Alarm Res
   // Interlock Alarm Res
   #O_IntlkResAlm := #IntlkResAlm;
END_REGION

REGION Network 30: **** 8 - Outputs **** Command High set
   // Command set
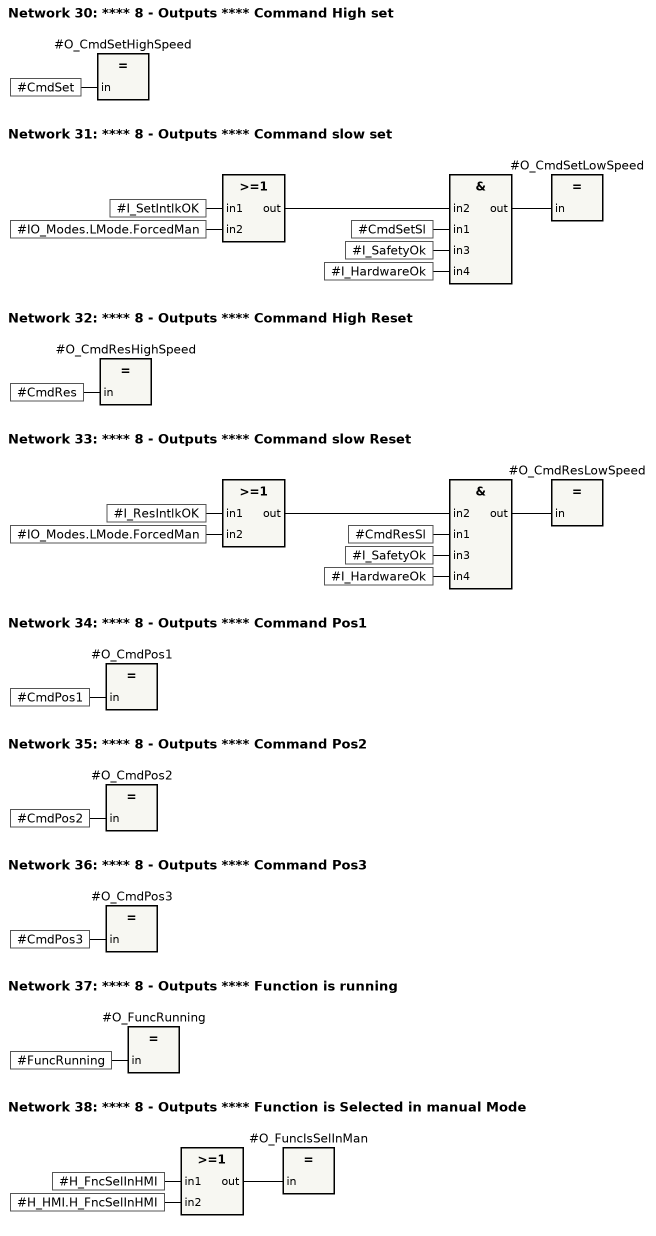
   #O_CmdSetHighSpeed := #CmdSet;
END_REGION

REGION Network 31: **** 8 - Outputs **** Command slow set
   // Command slow set
   #O_CmdSetLowSpeed := (#I_SetIntlkOK OR #IO_Modes.LMode.ForcedMan) AND #CmdSetSl AND #I_SafetyOk AND #I_HardwareOk;
END_REGION

REGION Network 32: **** 8 - Outputs **** Command High Reset
   // Command Reset
   #O_CmdResHighSpeed := #CmdRes;
END_REGION

REGION Network 33: **** 8 - Outputs **** Command slow Reset
   // Command slow Reset
   #O_CmdResLowSpeed := (#I_ResIntlkOK OR #IO_Modes.LMode.ForcedMan) AND #CmdResSl AND #I_SafetyOk AND #I_HardwareOk;
END_REGION

REGION Network 34: **** 8 - Outputs **** Command Pos1
   // Command Pos1
   #O_CmdPos1 := #CmdPos1;
END_REGION

REGION Network 35: **** 8 - Outputs **** Command Pos2
   // Command Pos2
   #O_CmdPos2 := #CmdPos2;
END_REGION

REGION Network 36: **** 8 - Outputs **** Command Pos3
   // Command Pos3
   #O_CmdPos3 := #CmdPos3;
END_REGION

REGION Network 37: **** 8 - Outputs **** Function is running
   // Function is running
   #O_FuncRunning := #FuncRunning;
END_REGION

REGION Network 38: **** 8 - Outputs **** Function is Selected in manual Mode
   // Function is Selected in manual Mode
   #O_FuncIsSelInMan := #H_FncSelInHMI OR #H_HMI.H_FncSelInHMI;
END_REGION

REGION Network 39: **** 8 - Outputs **** LED - Indication
   // LED - Indication
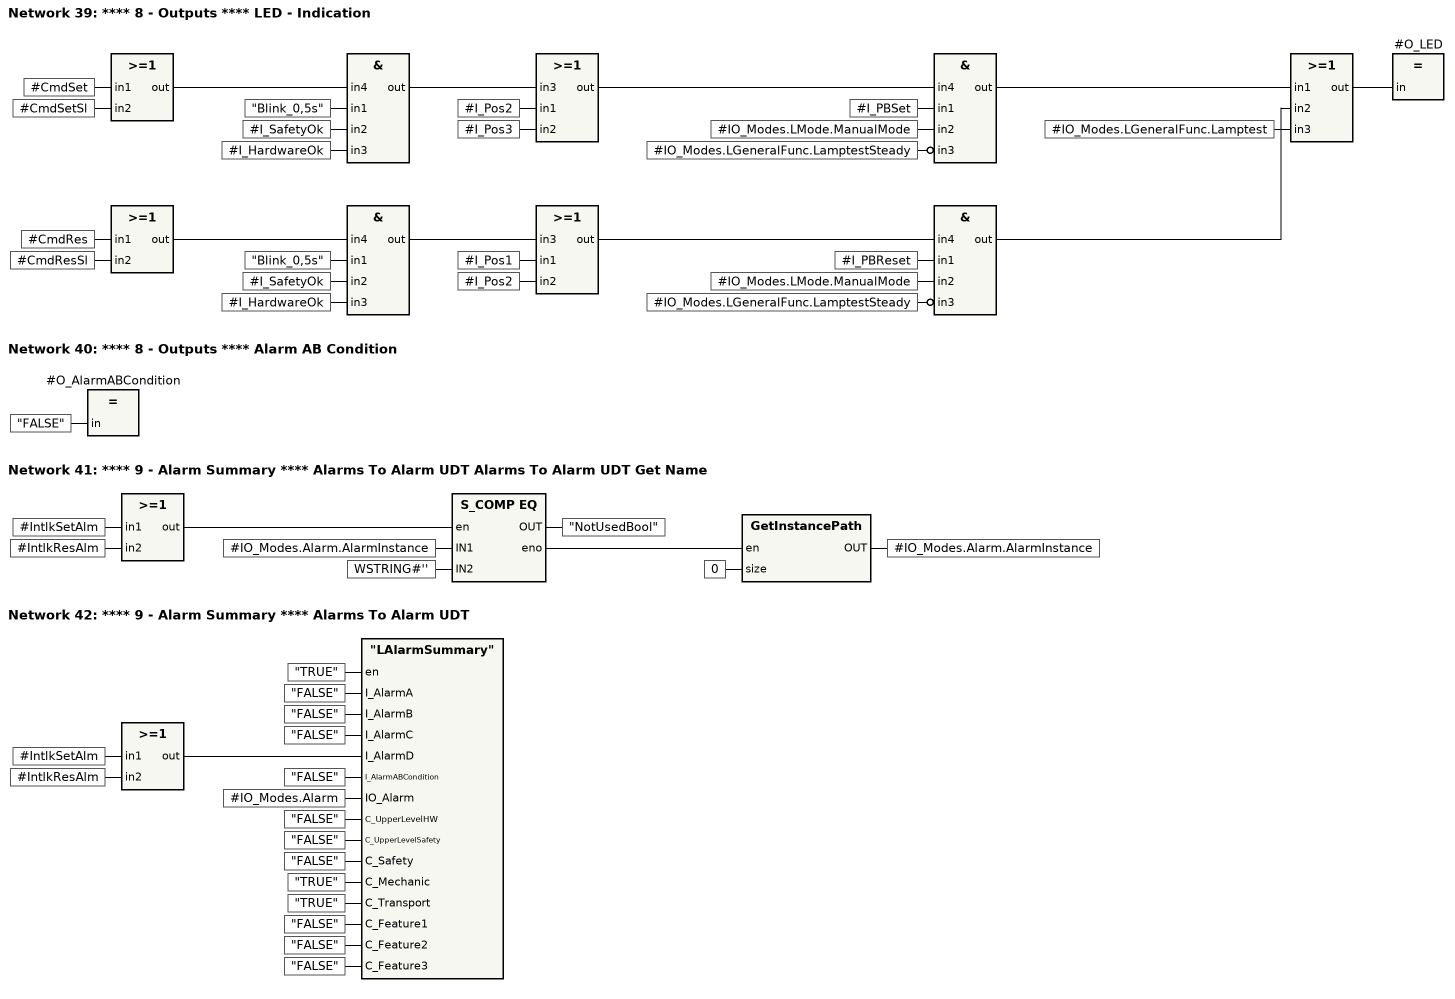
   #O_LED := ((((#CmdSet OR #CmdSetSl) AND "Blink_0,5s" AND #I_SafetyOk AND #I_HardwareOk) OR #I_Pos2 OR #I_Pos3) AND #I_PBSet AND #IO_Modes.LMode.ManualMode AND NOT #IO_Modes.LGeneralFunc.LamptestSteady) OR ((((#CmdRes OR #CmdResSl) AND "Blink_0,5s" AND #I_SafetyOk AND #I_HardwareOk) OR #I_Pos1 OR #I_Pos2) AND #I_PBReset AND #IO_Modes.LMode.ManualMode AND NOT #IO_Modes.LGeneralFunc.LamptestSteady) OR #IO_Modes.LGeneralFunc.Lamptest;
END_REGION

REGION Network 40: **** 8 - Outputs **** Alarm AB Condition
   // Alarm AB Condition
   #O_AlarmABCondition := "FALSE";
END_REGION

REGION Network 41: **** 9 - Alarm Summary **** Alarms To Alarm UDT Alarms To Alarm UDT Get Name
   // Alarms To Alarm UDT Alarms To Alarm UDT Get Name
   S_COMP(EN := #IntlkSetAlm OR #IntlkResAlm,
          IN1 := #IO_Modes.Alarm.AlarmInstance,
          IN2 := WSTRING#'',
          OUT => "NotUsedBool",
          ENO => #_w1);
   IF #_w1 THEN GetInstancePath(size := 0, OUT => #IO_Modes.Alarm.AlarmInstance); END_IF;
END_REGION

REGION Network 42: **** 9 - Alarm Summary **** Alarms To Alarm UDT
   // Alarms To Alarm UDT
   IF "TRUE" THEN
       "LAlarmSummary"(I_AlarmA := "FALSE",
                       I_AlarmB := "FALSE",
                       I_AlarmC := "FALSE",
                       I_AlarmD := #IntlkSetAlm OR #IntlkResAlm,
                       I_AlarmABCondition := "FALSE",
                       IO_Alarm := #IO_Modes.Alarm,
                       C_UpperLevelHW := "FALSE",
                       C_UpperLevelSafety := "FALSE",
                       C_Safety := "FALSE",
                       C_Mechanic := "TRUE",
                       C_Transport := "TRUE",
                       C_Feature1 := "FALSE",
                       C_Feature2 := "FALSE",
                       C_Feature3 := "FALSE");
   END_IF;
END_REGION
END_FUNCTION_BLOCK
